// TIA Portal V16 export
// export: Created 2023-10-30T22:43:54.7576289Z, ExportSetting WithDefaults, DisplayName Totally Integrated Automation Portal, DisplayVersion V16, DisplayName TIA Portal Version Control Interface, DisplayVersion V16, DisplayName TIA Portal Openness, DisplayVersion V16, DisplayName SINAMICS Startdrive Advanced, DisplayVersion V16, DisplayName SINAMICS Startdrive G130, G150, S120, S150, SINAMICS MV, S210, DisplayVersion V16, DisplayName SINAMICS Startdrive G110M, G120, G120C, G120D, G120P, DisplayVersion V16, DisplayName STEP 7 Professional, DisplayVersion V16, DisplayName STEP 7 Safety, DisplayVersion V16, DisplayName WinCC Professional, DisplayVersion V16
DATA_BLOCK "MB_CONFIG"   // DB9
{ S7_Optimized_Access := 'FALSE' }
VERSION : 0.1
// stored: AutoNumber true, DBAccessibleFromOPCUA true, IsOnlyStoredInLoadMemory false, IsWriteProtectedInAS false
   VAR
      Again : Bool;
      Req : Bool;
      Mb_Addr : UInt := 1;
      Mode : USInt := 0;
      Data_Addr : UDInt := 40001;
      Data_Len : UInt := 5;
      Done : Bool;
      Busy : Bool;
      Error : Bool;
      Status : Word;
      Error_Status : Word;
      "Step" : Int := 1;
   END_VAR
BEGIN
END_DATA_BLOCK
